Universal Robots URScript: custom_script_4.urscript

textmsg("Custom script 4...")
movej([0,1.57,-1.57,3.14,-1.57,1.57], a=1.4, v=1.05, t=0, r=0)
